(*******************************************************************************
                          protoc-gen-twincat V0.0.0.0                           
                  https://github.com/TcHaxx/protoc-gen-twincat                  
*******************************************************************************)
{attribute 'no-analysis'}
TYPE ST_SensorReading :
STRUCT
	value : LREAL;
	precision : REAL;
	timestamp : LINT;
END_STRUCT
END_TYPE

(* stored: Version 1.1.0.1
   DUT ST_SensorReading: Id cb0b1ae1-0037-47ab-9c08-dc0bb0d99e53 *)
